// TIA Portal V21 export
DATA_BLOCK "Dinamico"   // DB18
{ S7_Optimized_Access := 'TRUE' }
// stored: MemoryReserve 100
   VAR RETAIN
      K_Stazioni { S7_SetPoint := 'True'} : Array[0..8, 0..5] of Int;
      Hmi : Struct
         K_StazioneDaAggiungere : Int := 0;
         K_NumStazioneHmi : Int := 0;
         AggiungiStazione : Bool := FALSE;
      END_STRUCT;
   END_VAR
BEGIN
   K_Stazioni[0,0..5] := 0;
   K_Stazioni[1,0..5] := 0;
   K_Stazioni[2,0..5] := 0;
   K_Stazioni[3,0..5] := 0;
   K_Stazioni[4,0..5] := 0;
   K_Stazioni[5,0..5] := 0;
   K_Stazioni[6,0..5] := 0;
   K_Stazioni[7,0..5] := 0;
   K_Stazioni[8,0..5] := 0;
END_DATA_BLOCK
